FUNCTION_BLOCK FB_PositionStatePMPS2D
(*
    Proof of concept for a 2D pmps state mover
    This should illustrate how many more building blocks need to be added to reach the goal
    When finished, this should be usable as a function block in live PLCs, just pragma and add your enum
    Need to also make 1D, 3D, and non-pmps versions
    Known missing:
    - Some FFOs aren't here yet
    - Database reading isn't here yet
*)
VAR_IN_OUT
    stMotionStage1: DUT_MotionStage;
    astPositionStates1: ARRAY[1..GeneralConstants.MAX_STATES] OF DUT_PositionState;
    stMotionStage2: DUT_MotionStage;
    astPositionStates2: ARRAY[1..GeneralConstants.MAX_STATES] OF DUT_PositionState;
    fbFFHWO: FB_HardwareFFOutput;
    fbArbiter: FB_Arbiter;
END_VAR
VAR_INPUT
    nSetPoint: DINT;
    {attribute 'pytmc' := '
        pv: STATES
    '}
    // TODO does this need to split into inputs and outputs?
    stEpicsInputs: DUT_StatePMPSEpicsInterface;
END_VAR
VAR_OUTPUT
    nReadback: DINT;
END_VAR
VAR
    astAllMotors: ARRAY[1..2] OF DUT_MotionStage;
    astFullPositionStates: ARRAY[1..2, 1..GeneralConstants.MAX_STATES] OF DUT_PositionState;
    astDbStateParams: ARRAY[0..GeneralConstants.MAX_STATES] OF ST_DbStateParams;

    fbDB: FB_MotionReadPMPSDBND;
    fbBPTM: FB_MotionBPTM;
    fbLimits: FB_StatePMPSLimitsND;
    afbStateLimits: ARRAY[1..2] OF FB_StatePMPSLimits;
    fbMove: FB_PositionStateMoveND;
    afbMove: ARRAY[1..2] OF FB_PositionStateMove;
    fbRead: FB_PositionStateReadND;
    afbRead: ARRAY[1..2] OF FB_PositionStateRead;
END_VAR


// TODO if I assign like this here and invert at the end of the FB, does it work?
// Otherwise I need to use POINTER or REFERENCE
astAllMotors[1] := stMotionStage1;
astAllMotors[2] := stMotionStage2;

astFullPositionStates[1] := astPositionStates1;
astFullPositionStates[2] := astPositionStates2;

fbDB(
    astPositionState:=astFullPositionStates,
    astDbStateParams:=astDbStateParams,
    fbFFHWO:=fbFFHWO,
    sTransitionKey:=sTransitionKey,
    sDeviceName:=sDeviceName,
    bError=>,
    bArrayMismatchError=>,
);

fbBPTM(
    astMotionStage:=astAllMotors,
    fbArbiter:=fbArbiter,
    fbFFHWO:=fbFFHWO,
    stGoalParams:=stGoalParams,
    stTransParams:=stTransParams,
    bAtState:=bAtState,
    sDeviceName:=sDeviceName,
    tArbiterTimeout:=tArbiterTimeout,
    bMoveOnArbiterTimeout:=bMoveOnArbiterTimeout,
    bResetBPTMTimeout:=bResetBPTMTimeout,
    bTransitionAuthorized=>,
    bDone=>,
);

fbLimits(
    astMotionStage:=astAllMotors,
    astPositionState:=astFullPositionStates,
    afbStateLimits:=afbStateLimits,
    fbFFHWO:=fbFFHWO,
    nGoalStateIndex:=nGoalStateIndex,
    bArrayMismatchError=>,
);

fbMove(
    astMotionStage:=astAllMotors,
    astPositionState:=astCurrentGoalStates,
    afbPositionStateMove:=afbMove,
    bExecute:=bTimeToMove,
    bReset:=bTimeToReset,
    enumMotionRequest:=ENUM_MotionRequest.INTERRUPT,
    bAtState=>,
    bBusy=>,
    bDone=>,
    bError=>,
    nErrorCount=>,
    nShownError=>,
    nErrorID=>,
    sErrorMessage=>,
);

fbRead(
    astMotionStage:=astAllMotors,
    astPositionState:=astFullPositionStates,
    afbPositionStateRead:=afbRead,
    bKnownState=>,
    bMovingState=>,
    nPositionIndex=>,
    bArrayMismatchError=>,
);

// Need to update the global state of the motion DUTs
// See top of this FB
stMotionStage1 := astAllMotors[1];
stMotionStage2 := astAllMotors[2];

END_FUNCTION_BLOCK

(* stored: Version 1.1.0.1, ProductVersion 3.1.4022.18
   POU FB_PositionStatePMPS2D: Id {9dffd600-2d32-4e33-bb6b-8aab4cc29ee5}, SpecialFunc None *)
